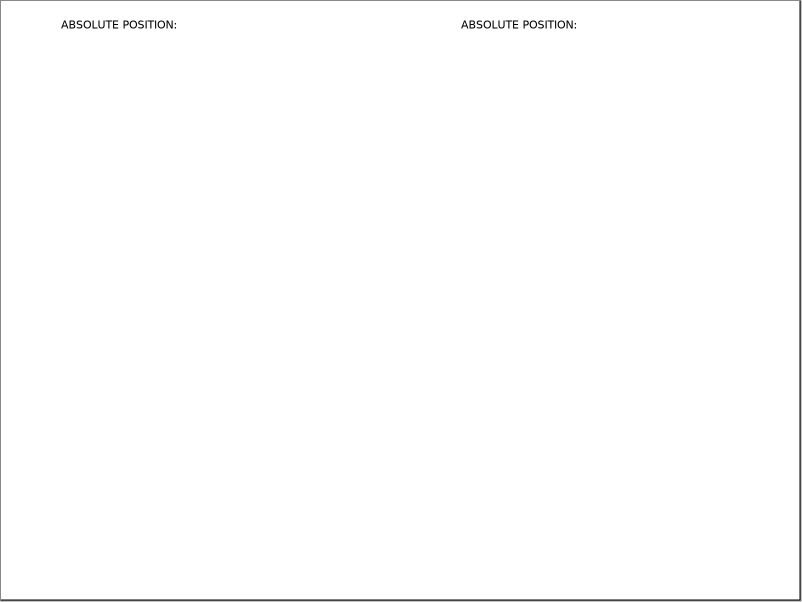
VISUALIZATION F50_Cam_Add  // 802x602
    Rectangle (0,0 800x600)
    Label (10,10 170x30), "ABSOLUTE POSITION:"
    Label (410,10 170x30), "ABSOLUTE POSITION:"
END_VISUALIZATION

(* stored: Version 1.1.0.1, ProductVersion 3.1.4022.7
   Visu F50_Cam_Add: Id {f362006f-daf1-49f5-9a17-d0a66f596296} *)
